Yaskawa INFORM job: S1.JBI

/JOB
//NAME S1
///FOLDERNAME INNE
//POS
///NPOS 0,0,6,0,0,0
///TOOL 0
///POSTYPE PULSE
///PULSE
EC00000=0,0
EC00001=1995323,0
EC00002=-1995282,0
EC00003=0,2782327
EC00004=0,-2782364
EC00005=0,0
//INST
///DATE 2023/10/04 15:16
///ATTR SC,RW,RJ
////FRAME ROBOT
///GROUP1 ST1
NOP
MOVJ EC00000 VJ=100.00
TIMER T=1.00
MOVJ EC00001 VJ=100.00
TIMER T=1.00
MOVJ EC00002 VJ=100.00
TIMER T=1.00
MOVJ EC00003 VJ=100.00
TIMER T=1.00
MOVJ EC00004 VJ=100.00
TIMER T=1.00
MOVJ EC00005 VJ=100.00
END
